Staubli VAL3: clkValve1.pgx

program clkValve1()
begin
  call toggleValve(1)
end
